PROGRAM prgGrid
VAR
	lrPowerGridkW		: LREAL;	//{#lynus.ag#()}
END_VAR

lrPowerGridkW := prgShelly.lrPowerCSTotalkW + prgShelly.lrPowerGarageTotalkW + prgShelly.lrPowerUVKellerTotalkW - prgPV.lrPowerPV;

END_PROGRAM

(* stored: Version 1.1.0.1, ProductVersion 3.1.4024.11
   POU prgGrid: Id {8baae4b7-808e-49f6-9066-8b3ec47f7a46}, SpecialFunc None *)
